// TIA Portal V20 export
DATA_BLOCK "DB_MainDoorManagement"   // DB96
// stored: InstanceOfName FB_MainDoorManagement, InstanceOfType FB
"FB_MainDoorManagement"
   // VAR
   //    FT_AxisDesactivated { S7_SetPoint := 'True'} : F_TRIG;
   //    sDoorNotLocked : Bool;
   //    sLockAutoFrontDoor : Bool;
   // END_VAR
BEGIN
END_DATA_BLOCK
